{attribute 'linkalways'} 
{attribute 'no_explicit_call' := 'This FB is a CLASS and must be accessed using methods or properties'}
{attribute 'enable_dynamic_creation'}
FUNCTION_BLOCK Node_F_VN_MedianElementElementwise_TcVnVector4_SINT EXTENDS VisionNode
VAR
    ipContainer : _ITcVnContainer;
    aMedian : _TcVnVector4_SINT;
    hrPrev : _HRESULT(S_OK);
    hresult : _HRESULT(S_OK);
END_VAR

METHOD PUBLIC  Clone : I_Node
VAR
	pNode : POINTER TO Node_F_VN_MedianElementElementwise_TcVnVector4_SINT;
END_VAR
pNode := __NEW(Node_F_VN_MedianElementElementwise_TcVnVector4_SINT);
Clone := pNode^;
END_METHOD

METHOD FB_init : BOOL
VAR_INPUT
	bInitRetains : BOOL; // if TRUE, the retain variables are initialized (warm start / cold start)
	bInCopyCode : BOOL;  // if TRUE, the instance afterwards gets moved into the copy code (online change)
END_VAR
AddInput('ipContainer', ipContainer);
AddInput('aMedian', aMedian);
AddInput('hrPrev', hrPrev);
AddOutput('ipContainer', ipContainer);
AddOutput('hresult',hresult);
END_METHOD

METHOD PROTECTED OnExecute : HRESULT
hresult.Value := F_VN_MedianElementElementwise_TcVnVector4_SINT(
    ipContainer := ipContainer.Value,
    aMedian := aMedian.Value,
    hrPrev:= hrPrev.Value);
END_METHOD

METHOD PUBLIC PreExecutionCheck
VAR_INPUT
	Check : I_PreExecutionChecks;
END_VAR
Check.IsTrue(ipContainer.IsValid, 'ipContainer must be a valid container');
END_METHOD

END_FUNCTION_BLOCK

(* stored: Version 1.1.0.1, ProductVersion 3.1.4024.13
   POU Node_F_VN_MedianElementElementwise_TcVnVector4_SINT: Id {26f323f7-f915-49b6-9a02-17ff0892277d}, SpecialFunc None
   Folder Constructor: Id {1023a05b-5361-4605-b2d2-dd4db631054c}
   Method Clone: Id {ea381945-ea89-4296-9571-0d939c24cfbc}
   Method FB_init: Id {576dfc2e-c908-4afc-a6e1-0b82b4797950}
   Method OnExecute: Id {915ce213-6a9e-436e-a8eb-fa0643cdce7d}
   Method PreExecutionCheck: Id {d43c5db3-7de7-434d-8481-241d3c3fe420} *)
